// TwinCAT 3 PLC project AdsClient
// ProgramVersion: 3.1.4026.21
// libraries:
//   Tc2_MC2, * (Beckhoff Automation GmbH)
//   Tc2_Standard, * (Beckhoff Automation GmbH)
//   Tc2_System, * (Beckhoff Automation GmbH)
// project tree:
//   / PlcTask.TcTTO
//   POUs/ MAIN.TcPOU
// real-time tasks:
//   TASK PlcTask: cycle T#10ms, priority 20, ADS port 350
// motion (NC):
//   TASK NC-Task 1 SAF: cycle T#2ms, priority 4, ADS port 501
//   TASK NC-Task 1 SVB: cycle T#10ms, priority 8, ADS port 511
//   AXIS Axis1 (id 1)
//     OtherSettings: AllowMotionCmdToSlave=true
//     encoder EncType=1
//     drive DrvType=5
//       Analog: TorqueSetpointScale=10, ScaleFactorActTorque=0.1
//     controller CtrType=1
//       CtrPara: PriorControlFactor=1
//         Observer: BandWidth=20
// variable links:
//   (this object) <-> NC-Task 1 SAF/Axes/Axis1
//     PlcTask Inputs/MAIN.axis1.NcToPlc <-> Outputs/ToPlc
//     PlcTask Outputs/MAIN.axis1.PlcToNc <-> Inputs/FromPlc

CONFIGURATION AdsClient
    RESOURCE PLC ON TwinCAT3
        TASK PlcTask(INTERVAL := T#10ms, PRIORITY := 20);
        PROGRAM MAIN WITH PlcTask : MAIN;
    END_RESOURCE
END_CONFIGURATION

// ---- POUs/MAIN.TcPOU
PROGRAM MAIN
VAR
	{attribute 'TcNcAxis' := 'Axis1'}
	axis1		: AXIS_REF;
	mcPower		: MC_Power;
	mcReset		: MC_Reset;
	mcHalt		: MC_Halt;
	mcVelocity	: MC_MoveVelocity;
	
	powerOnAxis		: BOOL;
	resetAxis		: BOOL;
	moveAxis		: BOOL;
	moveVelocity	: LREAL := 100.0;
	axisPosition	: LREAL;
END_VAR

mcVelocity(
	Axis:= axis1, 
	Execute:= moveAxis AND powerOnAxis, 
	Velocity:= moveVelocity 
);

mcHalt(
	Axis:= axis1, 
	Execute:= NOT moveAxis
);

mcReset(
	Axis:= axis1, 
	Execute:= resetAxis
);

mcPower(
	Axis:= axis1, 
	Enable:= powerOnAxis, 
	Enable_Positive:= powerOnAxis, 
	Enable_Negative:= powerOnAxis
);

axisPosition := axis1.NcToPlc.ActPos;

END_PROGRAM
